PROGRAM Motion01
VAR
	MC_Power_0				: MC_Power;
	Axis01					: AXIS_REF;
	A1_En					: BOOL;
	MC_Power_1				: MC_Power;
	Axis02					: AXIS_REF;
	A2_En					: BOOL;
	MC_MoveVelocity_0		: MC_MoveVelocity;
	MC_MoveVelocity_1		: MC_MoveVelocity;
	V1_En					: BOOL;
	V2_En					: BOOL;
	MC_Stop_0				: MC_Stop;
	V1_Stp					: BOOL;
	MC_Stop_1				: MC_Stop;
	V2_Stp					: BOOL;
	V1						: LREAL;
	V2						: LREAL;
	MC_Jog_0				: MC_Jog;
	Jog_For					: BOOL;
	MC_MoveRelative_0		: MC_MoveRelative;
	Move_Do					: BOOL;
	MC_SetPosition_0		: MC_SetPosition;
	Set_Do					: BOOL;
	Power_Do				: BOOL;
	MC_Jog_1				: MC_Jog;
	MC_MoveRelative_1		: MC_MoveRelative;
	MC_SetPosition_1		: MC_SetPosition;
	Stop_Do					: BOOL;
	MC_Reset_0				: MC_Reset;
	Reset_Do				: BOOL;
	MC_Reset_1				: MC_Reset;
	MC_GearIn_0				: MC_GearIn;
	MC_GearOut_0			: MC_GearOut;
	Gearin_Do				: BOOL;
	Gearout_Do				: BOOL;
	MC_Home_0				: MC_Home;
	Home_Do					: BOOL;
	Sensor					: BOOL;
	MC_CamIn_0				: MC_CamIn;
	Cam_Do					: BOOL;
	MC_CamOut_0				: MC_CamOut;
	Camout_Do				: BOOL;
END_VAR

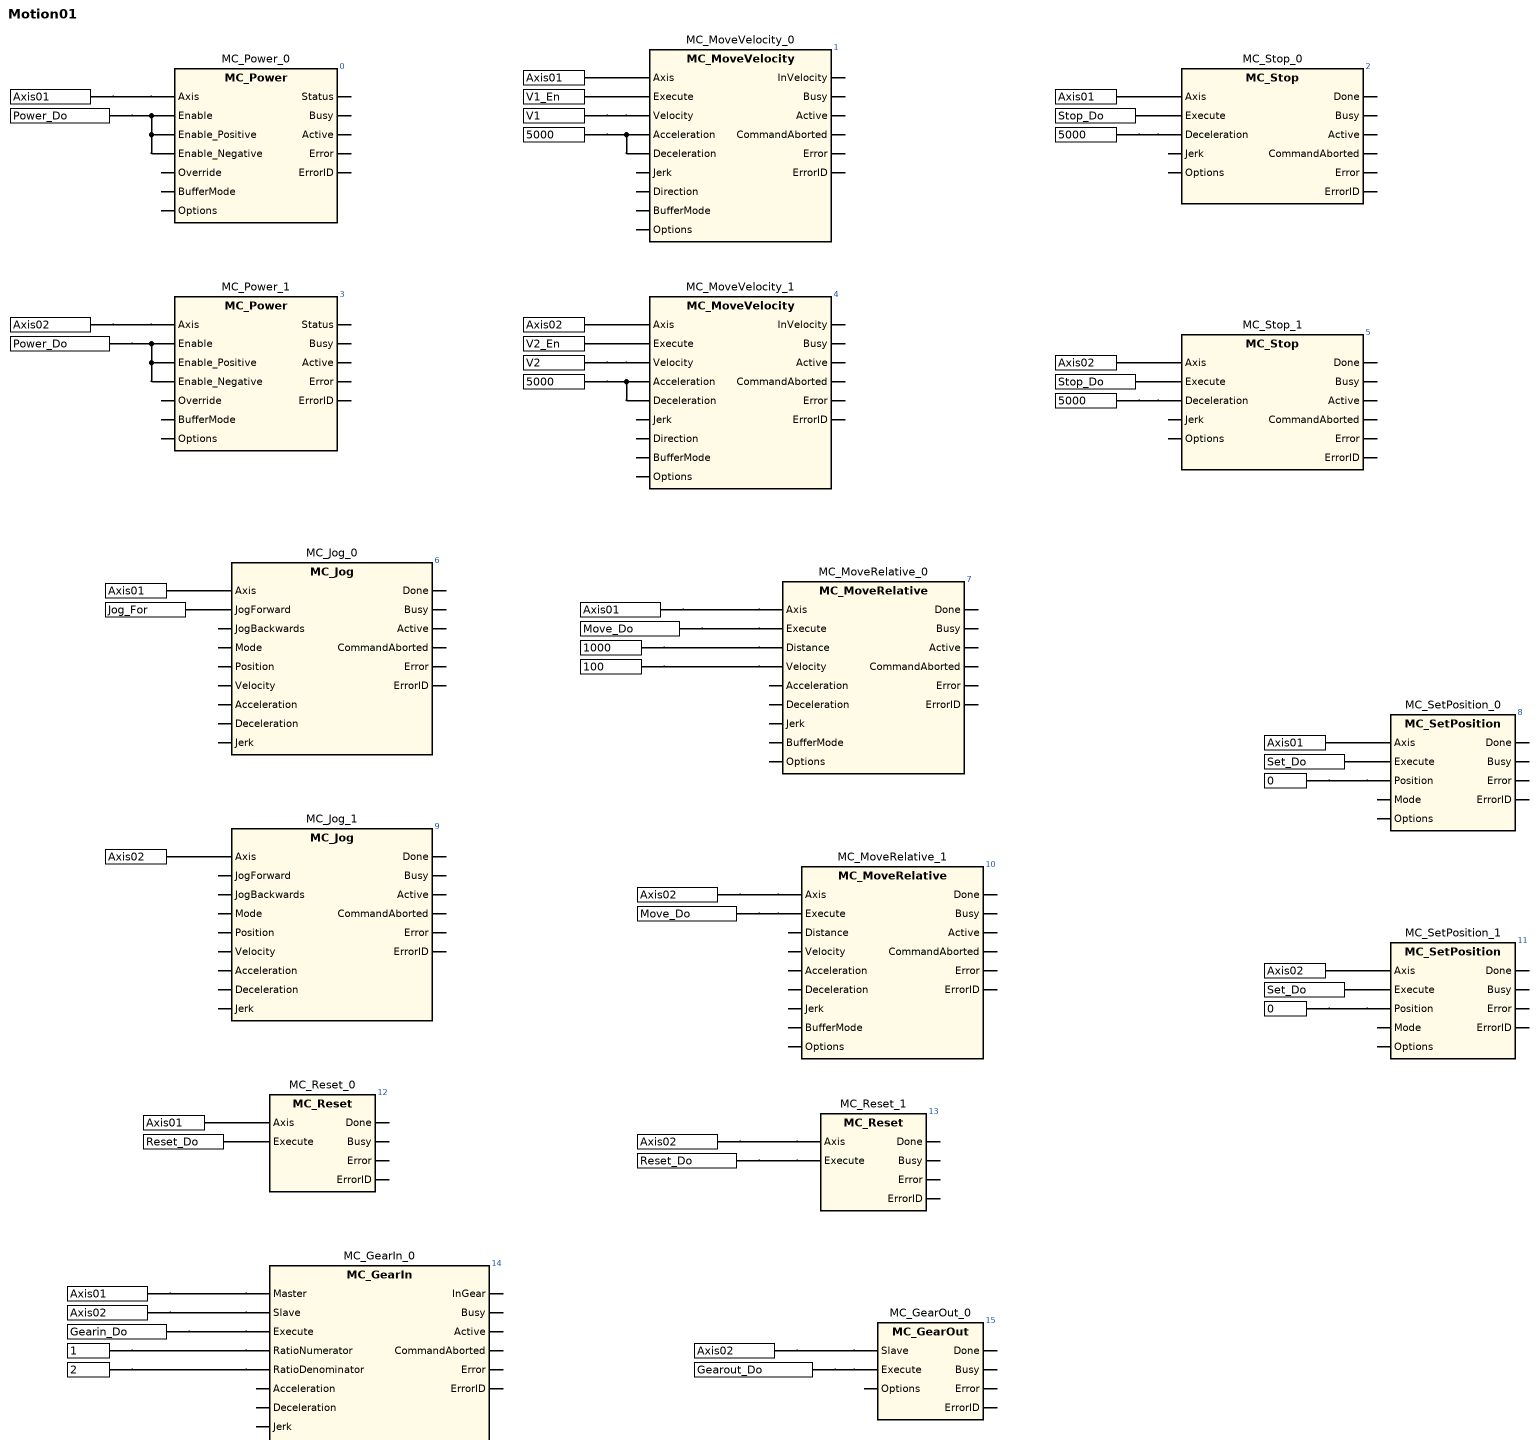
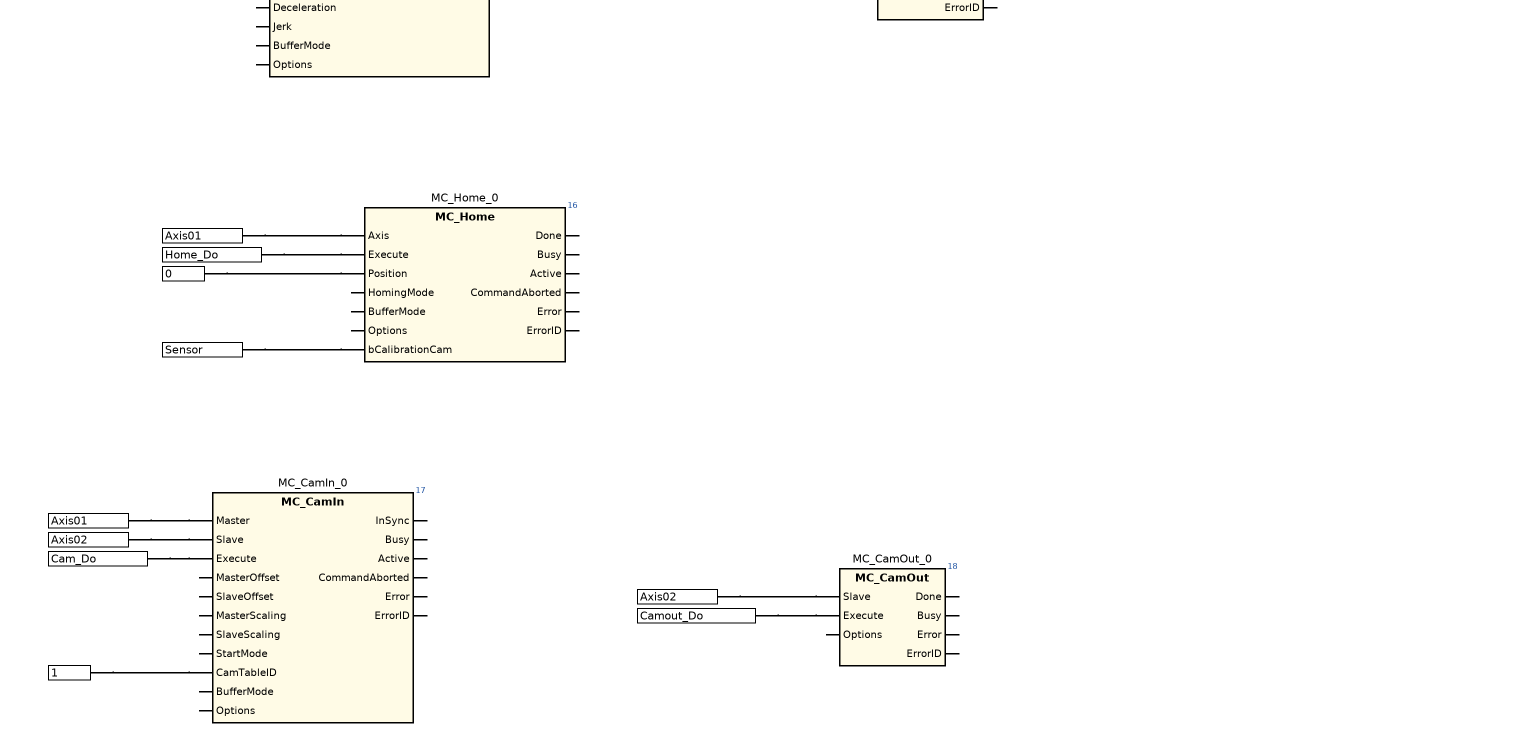
MC_Power_0(Axis := Axis01, Enable := Power_Do, Enable_Positive := Power_Do, Enable_Negative := Power_Do); // MC_Power
MC_MoveVelocity_0(
    Axis := Axis01,
    Execute := V1_En,
    Velocity := V1,
    Acceleration := 5000,
    Deceleration := 5000); // MC_MoveVelocity
MC_Stop_0(Axis := Axis01, Execute := Stop_Do, Deceleration := 5000); // MC_Stop
MC_Power_1(Axis := Axis02, Enable := Power_Do, Enable_Positive := Power_Do, Enable_Negative := Power_Do); // MC_Power
MC_MoveVelocity_1(
    Axis := Axis02,
    Execute := V2_En,
    Velocity := V2,
    Acceleration := 5000,
    Deceleration := 5000); // MC_MoveVelocity
MC_Stop_1(Axis := Axis02, Execute := Stop_Do, Deceleration := 5000); // MC_Stop
MC_Jog_0(Axis := Axis01, JogForward := Jog_For); // MC_Jog
MC_MoveRelative_0(Axis := Axis01, Execute := Move_Do, Distance := 1000, Velocity := 100); // MC_MoveRelative
MC_SetPosition_0(Axis := Axis01, Execute := Set_Do, Position := 0); // MC_SetPosition
MC_Jog_1(Axis := Axis02); // MC_Jog
MC_MoveRelative_1(Axis := Axis02, Execute := Move_Do); // MC_MoveRelative
MC_SetPosition_1(Axis := Axis02, Execute := Set_Do, Position := 0); // MC_SetPosition
MC_Reset_0(Axis := Axis01, Execute := Reset_Do); // MC_Reset
MC_Reset_1(Axis := Axis02, Execute := Reset_Do); // MC_Reset
MC_GearIn_0(
    Master := Axis01,
    Slave := Axis02,
    Execute := Gearin_Do,
    RatioNumerator := 1,
    RatioDenominator := 2); // MC_GearIn
MC_GearOut_0(Slave := Axis02, Execute := Gearout_Do); // MC_GearOut
MC_Home_0(Axis := Axis01, Execute := Home_Do, Position := 0, bCalibrationCam := Sensor); // MC_Home
MC_CamIn_0(Master := Axis01, Slave := Axis02, Execute := Cam_Do, CamTableID := 1); // MC_CamIn
MC_CamOut_0(Slave := Axis02, Execute := Camout_Do); // MC_CamOut

END_PROGRAM

(* stored: Version 1.1.0.1, ProductVersion 3.1.4024.10
   POU Motion01: Id {2d610003-814f-490e-81a1-846bf07cfdea}, SpecialFunc None *)
